(*~
	<docu>
		<summary>
			Root construction container, provides context information for <c>TcoObjects</c> declared within its scope.
			This function block is ```abstract``` and cannot be instantiated. 
			Use <see cref="TcoContext.PlcTcoContext.Run()"/> to run this context, ```Run``` method must be called only once per Plc's Task cycle.
			Several 'TcoContext' instances can be declared and called inside one TwinCAT PlcTask, but only once per plc cycle. The instance should not be accessed from several Twincat PlcTasks.
			Default implemenation of the 'TcoContext' allows its child members access properties <see cref="TcoContext.PlcTcoContext.StartCycleCount()"/> and <see cref="TcoContext.PlcTcoContext.EndCycleCount()"/>.\			 			 			
			<note type="tip">
				 A <c>TcoContext</c> can contain objects, components and PLC logic of one independent station of the machine, while the another one can cover the same for another station.			
			</note>
			<remarks>			
				<note type="tip">
					TwinCAT PlcTask and <see cref="TcoTask.PlcTcoTask()"/> refer to two different concepts. 
				</note>
			</remarks>
		</summary>	
		<example>
			Declaration part of the 'TcoContext' example. 
		</example>
		<example>
				[!code-pas[Main](~/../TcOpen/src/TcoApplicationExamples/XaeAppExamples/PlcAppExamples/POUs/Context/VitoCorleone_Context.TcPOU?name=ContextExampleDeclarations)]
		</example>
		<example>
			Implementation part of the 'TcoContext' example.
		</example>
		<example>
				[!code-pas[Main](~/../TcOpen/src/TcoApplicationExamples/XaeAppExamples/PlcAppExamples/POUs/Context/VitoCorleone_Context.TcPOU?name=ContextExampleCode)]
		</example>
	</docu>	
~*)
FUNCTION_BLOCK PUBLIC ABSTRACT TcoContext IMPLEMENTS ITcoContext
VAR
	(*~
		<docu>
			<summary>
				Identity of this <c>TcoContext</c>.
				This variable is used in the higher level packages. 
				Allows for identification of the specific context in SCADA like applications.	  
			</summary>			
		</docu>	
	~*)
	{attribute clr [RenderIgnore()]}
	{attribute clr [ReadOnly()]}
	_Identity : ULINT;
	{attribute clr [ReadOnly()]}
	_startCycleCount : ULINT;
	{attribute clr [ReadOnly()]}
	_endCycleCount : ULINT;
	_messagingLevel : eMessageCategory;
	{attribute clr [ReadOnly()]}
	_rtc : TcoRtc;
	{attribute clr [RenderIgnore()]}
    _settings : TcoContextEnvironment;	
END_VAR

(*~
	<docu>
		<summary>
			This method is called implicitly at the entry point of this context (<see cref="TcoContext.PlcTcoContext.Run()"/>).
			<remarks>			
				<note type="important">
					Do not call this method explicitly!
				</note>
			</remarks>
		</summary>			
	</docu>	
~*)
METHOD INTERNAL FINAL Close
_endCycleCount := _startCycleCount;
THIS^.PostRun();
END_METHOD

(*~
	<docu>
		<summary>
			Returns reference to this instance of the <see cref="TcoContext.PlcTcoContext()"/>.
		</summary>			
	</docu>	
~*)
PROPERTY Context : ITcoContext
GET
Context := THIS^;
END_GET
END_PROPERTY

(*~
	<docu>
		<summary>
		    Gets the value of the counter incrememented by '1' at the end of each execution of this <see cref="TcoContext.PlcTcoContext()"/>.			
		</summary>			
	</docu>	
~*)
PROPERTY EndCycleCount : ULINT
GET
EndCycleCount := _endCycleCount;
END_GET
END_PROPERTY

PROPERTY Environment : ITcoContextEnvironment
GET
Environment := _settings;
END_GET
END_PROPERTY

METHOD FB_init : BOOL
VAR_INPUT
	bInitRetains : BOOL; // if TRUE, the retain variables are initialized (warm start / cold start)
	bInCopyCode : BOOL;  // if TRUE, the instance afterwards gets moved into the copy code (online change)
END_VAR
_Identity := ADR(THIS^);
END_METHOD

(*~
	<docu>
		<summary>
			Returns the identity of this <see cref ="TcoContext.PlcTcoContext()"/>. 
			This value is assigned when instantiated and cannot be changed at runtime.
			This member is used in the higher level packages.  
		</summary>			
	</docu>	
~*)
PROPERTY Identity : ULINT
GET
Identity := _Identity;
END_GET
END_PROPERTY

(*~
	<docu>
		<summary>
			Main method of the TcoContext. This is the entry point of any control logic that belongs to this context. 
			The call of this method is ensured by calling the <c>InstanceName.Run()</c> method, and it must not be called explicitly.
			This method is abstract, and it must be overridden in derived block.
		</summary>
	</docu>
~*)
METHOD PROTECTED ABSTRACT Main
END_METHOD

(*~
	<docu>
		<summary>
			This method is called implicitly at the entry point of this context (<see cref="TcoContext.PlcTcoContext.Run()"/>).
			<remarks>			
				<note type="important">
					Do not call this method explicitly.
				</note>
			</remarks>
		</summary>			
	</docu>	
~*)
METHOD INTERNAL FINAL Open
THIS^.PriorRun();
_startCycleCount := _startCycleCount + 1;
_rtc.Update();
END_METHOD

METHOD PROTECTED PostRun
END_METHOD

METHOD PROTECTED PriorRun
END_METHOD

PROPERTY Rtc : ITcoRtc
GET
Rtc := _rtc;
END_GET
END_PROPERTY

METHOD RtcSynchronize  : REFERENCE TO TcoContext
VAR_INPUT
	inDoSynch				:	BOOL;
	inSyncAmsId				:	STRING;
	inSyncPeriod			:	UINT; 
END_VAR
VAR
	_RtcSynchParams						:	RtcSynchParams;			
END_VAR
_RtcSynchParams.doSynch					:=	inDoSynch;
_RtcSynchParams.syncAmsId				:=	inSyncAmsId;
_RtcSynchParams.syncPeriod				:=	inSyncPeriod;
_RtcSynchParams.synchContextIdentity	:=	THIS^._Identity;
RtcPrg.Synchronize(_RtcSynchParams);
RtcSynchronize REF= THIS^;
END_METHOD

(*~
	<docu>
		<summary>
			<para>
				This method executes of this context. It provided correct order of execution order of inner methods. Any logic of this context must be called within <see cref="TcoContext.PlcTcoContext.Main()"/>
				method. This method is final, so it cannot be overriden. The <c>InstanceName.Run()</c> needs to be called cyclically.
			</para>
		</summary>			
	</docu>	
~*)
METHOD PUBLIC FINAL Run
THIS^.Open();
THIS^.Main();
THIS^.Close();
END_METHOD

(*~
	<docu>
		<summary>
		    Gets number of executions of this context. Value of this property is incremented by '1' at the beginning of the <see cref="TcoContext.PlcTcoContext()"/>. 			 			
		</summary>			
	</docu>	
~*)
PROPERTY StartCycleCount : ULINT
GET
StartCycleCount := _startCycleCount;
END_GET
END_PROPERTY

END_FUNCTION_BLOCK

(* stored: Version 1.1.0.1, ProductVersion 3.1.4024.6
   POU TcoContext: Id {55d37a51-70a7-4749-9f28-95ccbcaee495}, SpecialFunc None
   Method Close: Id {75878743-2aed-4461-9dcd-3dcede9d89a5}
   Property Context: Id {63063553-badc-4ce8-a8c6-8619f5f133f3}
   Get Get: Id {892fc39b-0726-4b20-b0e0-f4be7b7e4106}
   Property EndCycleCount: Id {4bd5fb2b-81cd-4c36-8e15-26aba6b66c8a}
   Get Get: Id {095042f2-367c-44fe-aa5f-66cbd722b7e1}
   Property Environment: Id {b26311d8-ac58-0fb2-3664-3d88502e5497}
   Get Get: Id {0d0a9027-69a3-091e-3f34-9615f510e71b}
   Method FB_init: Id {589fd291-1ab8-4b98-a0a8-8d493e4b98c7}
   Property Identity: Id {a551eec9-c5bd-4df5-9bc0-f8e8eaa3edde}
   Get Get: Id {af84927a-5c14-4bee-90d2-b1f9bf5c7a59}
   Method Main: Id {a4678500-dacf-4449-bf3c-2b4f4414d6a6}
   Method Open: Id {d862846f-7f33-47b7-aa0a-9f3ebf516821}
   Method PostRun: Id {cc3ded61-78cb-0c12-3071-9c305dc097e3}
   Method PriorRun: Id {48b3abea-36b3-0d8f-1718-3531af00fe19}
   Property Rtc: Id {0e8903d2-e271-0e74-274a-b8795daab1b3}
   Get Get: Id {2d224feb-78f3-050e-2237-96bc8473a6fe}
   Method RtcSynchronize: Id {fdad5da4-2f47-075c-1134-913896442d7c}
   Method Run: Id {c20d2d3c-fd63-4a1d-8862-cb4f91ebaf8c}
   Property StartCycleCount: Id {bfc0527d-ea91-4a81-9e56-7fd6b0f76c09}
   Get Get: Id {72057c13-7a51-41fe-9542-bf3438a07393} *)
